TYPE (* Typedef of the ISO CF/user information data array *)
  (* Version 1.0, 2025-09-04, franz *)
  PACKAGE isobus;
  CF_NAME_T : STRUCT
    data : ARRAY [0..7] OF BYTE := [16#FF, 16#FF, 16#FF, 16#FF, 16#FF, 16#FF, 16#FF, 16#FF];
  END_STRUCT;
END_TYPE
